(* PLC project CoDeSys External Library Template, WAGO e!COCKPIT e!COCKPIT, author 3S - Smart Software Solutions GmbH *)
(* stored: creationDateTime 2019-10-29T12:22:40.4932442, version 3.5.5.30, modificationDateTime 2019-10-24T14:40:07.960949, organization 3S - Smart Software Solutions GmbH *)
(* Library project template with all possible element types, docu and a sample project structure *)

(* values of enumPPPSWezelClimatixPOL63xTrybPracy: Auto: Tryb pracy automatycznej; OchronaBudynku: Tryb utrzymania minimalnych nastaw dla ochrony budynku; Ekonomiczny: Tryb Ekonomiczny; Komfort: Tryb komfortu; ReczneWylaczenie: Ręczne, lokalne wyłączenie węzła *)

(* Autor: Paweł Kąkol, 2018-09-03-PK Prawa majątkowe: Solwena Sp. z o.o., Aktualizacje: Opis: enum służy do obsługi Trybów pracy fb węzła Climatix POL63x na budynkach PPP Sopot (ENGIE) *)
{attribute 'qualified_only'}
{attribute 'strict'}
TYPE enumPPPSWezelClimatixPOL63xTrybPracy : (Auto := 0, OchronaBudynku := 1, Ekonomiczny := 2, Komfort := 3, ReczneWylaczenie := 4);
END_TYPE
